PROGRAM P_Demo_FB_HVACPersistentDataHandling
VAR
    fb : FB_HVACPersistentDataHandling;                            // 被演示 FB 实例
    sNETID_in : T_AmsNetId ;
    TMOUT_in : TIME := T#0S;
    ePersistentMode_in : E_PersistentMode ;
    udiStatus_out : UDINT;
    iPersistCount_out : INT;
    bDone_out : BOOL;
    bBusy_out : BOOL;
    bError_out : BOOL;
    udiErrorID_out : UDINT;
END_VAR

// ============================================================================
// Tc2_HVAC.FB_HVACPersistentDataHandling 演示程序
// ============================================================================
// 场景：把本 FB 实例化到一个 PLC 程序里，每周期单次调用；按需要把 VAR_INPUT 与
//       VAR_IN_OUT 接到工程信号；VAR_OUTPUT 写入对应监视变量。
// 价值：使用本 FB 比手写状态机 / 控制算法节省大量代码；与 Tc2_HVAC 体系内其它 FB
//       直接对接，命名 / 持久化 / 模式仲裁等约定一致。具体语义见 FB_HVACPersistentDataHandling.md 主文档。
// 验证步骤：
//   1. 右键 PLC 项目下 POUs 文件夹 → Add → Existing Item → 选本 .TcPOU 文件
//   2. 引用 Tc2_HVAC（References → Add library）
//   3. 编译 → 登录 → 运行
//   4. 在线写各 *_in 输入信号触发 FB；在线 monitor *_out 引脚观察状态
// ============================================================================

fb(
    sNETID := sNETID_in,
    TMOUT := TMOUT_in,
    ePersistentMode := ePersistentMode_in,
    udiStatus => udiStatus_out,
    iPersistCount => iPersistCount_out,
    bDone => bDone_out,
    bBusy => bBusy_out,
    bError => bError_out,
    udiErrorID => udiErrorID_out
);

END_PROGRAM

(* stored: Version 1.1.0.1, ProductVersion 3.1.4024.5
   POU P_Demo_FB_HVACPersistentDataHandling: Id {bfab022c-668a-5b5a-ad72-2127060284c7}, SpecialFunc None *)
